{attribute 'strict'}
TYPE E_KAnalogMeasure_States : 
( 
	KANALOGMEASURE_DISABLED,	
	KANALOGMEASURE_ENABLING,
	KANALOGMEASURE_READY,
	KANALOGMEASURE_ERROR
)BYTE;
END_TYPE

(* stored: Version 1.1.0.1, ProductVersion 3.1.4024.9
   DUT E_KAnalogMeasure_States: Id {ebfd1164-ecb8-4db5-8795-ba30c556f59a} *)
